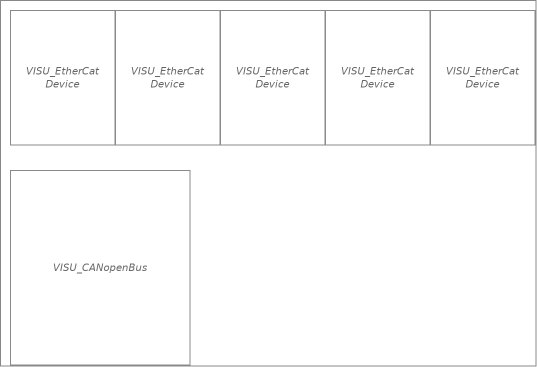
VISUALIZATION VISU_M3IO  // 537x367
VAR_IN_OUT	
    ref : M3IO;
    widget : M3IOWidget;
END_VAR
    Frame (430,10 105x135)
        shows VISU_EtherCatDevice(device := ref.parts.slot4, widget := widget.slot4)
    Frame (10,10 105x135)
        shows VISU_EtherCatDevice(device := ref.parts.coupler, widget := widget.coupler)
    Frame (115,10 105x135)
        shows VISU_EtherCatDevice(device := ref.parts.slot1, widget := widget.slot1)
    Frame (220,10 105x135)
        shows VISU_EtherCatDevice(device := ref.parts.slot2, widget := widget.slot2)
    Frame (325,10 105x135)
        shows VISU_EtherCatDevice(device := ref.parts.slot3, widget := widget.slot3)
    Frame (10,170 180x195)
        shows VISU_CANopenBus(ref := ref.parts.canOpenBus, widget := widget.canOpenBus)
END_VISUALIZATION

(* stored: Version 1.1.0.1, ProductVersion 3.1.4019.2
   Visu VISU_M3IO: Id {0962238c-4fcd-4e0f-8c0b-d04287c29818} *)
